FUNCTION_BLOCK IO_force
VAR_INPUT
	Raw_IO : BOOL;
END_VAR

VAR_OUTPUT
	Out : BOOL;
END_VAR

VAR
	ForceEnable : BOOL;
	ForceStatus : BOOL;
END_VAR

IF NOT ForceEnable THEN
	OUT := Raw_IO;
ELSE
	OUT := ForceStatus;
END_IF

END_FUNCTION_BLOCK

(* stored: Version 1.1.0.1, ProductVersion 3.1.4024.15
   POU IO_force: Id {56dfec2a-c0c6-4c6e-a8ee-f1954436e310}, SpecialFunc None *)
